FUNCTION SubtractionFunction : REAL
VAR_INPUT
	i_rValueA : REAL;
	i_rValueB : REAL;
VAR
END_VAR

SubtractionFunction := i_rValueA - i_rValueB;

END_FUNCTION

(* stored: Version 1.1.0.1, ProductVersion 3.1.4022.12
   POU SubtractionFunction: Id {e59e90e6-f992-4ed9-a990-96ffb17f3ff5}, SpecialFunc None *)
